// TIA Portal V20 export
DATA_BLOCK "DB_TX"   // DB12
{ S7_Optimized_Access := 'FALSE' }
   VAR
      Lifebit : Bool;
      Curing_in_auto_mode : Bool;
      Curing_in_operation : Bool;
      Curing_in_fault : Bool;
      Circulation_in_operaton : Bool;
      Heating_in_operation : Bool;
      Exhaust_Ventilator_in_operation : Bool;
      Doors_in_auto_mode : Bool;
      Door_1_is_open : Bool;
      Door_1_is_closed : Bool;
      Door_2_is_open : Bool;
      Door_2_is_closed : Bool;
      Door_3_is_open : Bool;
      Door_3_is_closed : Bool;
      Actual_Temperature : Int;
      Actual_Humidity : Int;
   END_VAR
BEGIN
END_DATA_BLOCK
